// Mitsubishi GX Works2 project: 알람 터치스크린   PLC: Q02/Q02H

PROGRAM MAIN
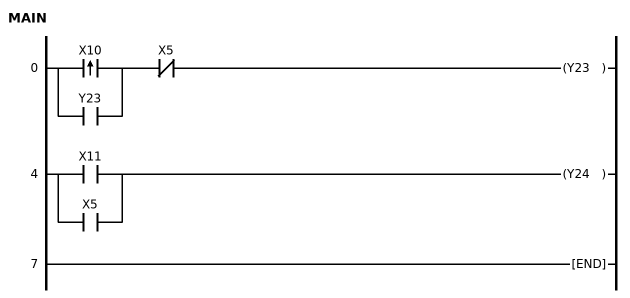
0     LDP     X10
      OR      Y23
      ANI     X5
      OUT     Y23
4     LD      X11
      OR      X5
      OUT     Y24
7     END
END_PROGRAM

PROGRAM HMI
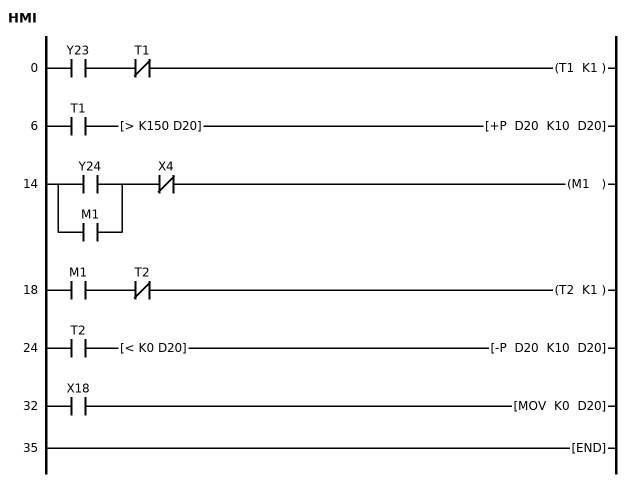
0     LD      Y23
      ANI     T1
      OUT     T1 K1
6     LD      T1
      AND>    K150 D20
      +P      D20 K10 D20
14    LD      Y24
      OR      M1
      ANI     X4
      OUT     M1
18    LD      M1
      ANI     T2
      OUT     T2 K1
24    LD      T2
      AND<    K0 D20
      -P      D20 K10 D20
32    LD      X18
      MOV     K0 D20
35    END
END_PROGRAM

PROGRAM ALARM
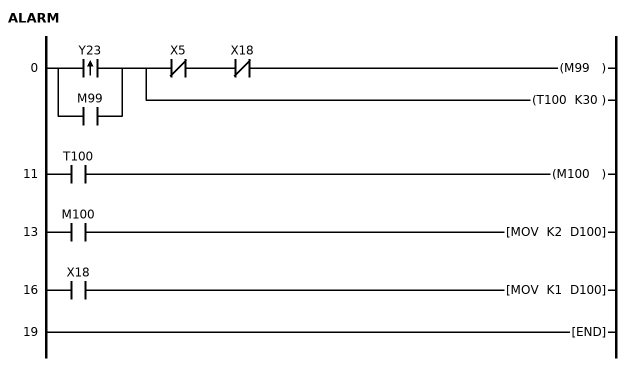
0     LDP     Y23
      OR      M99
      MPS
      ANI     X5
      ANI     X18
      OUT     M99
      MPP
      OUT     T100 K30
11    LD      T100
      OUT     M100
13    LD      M100
      MOV     K2 D100
16    LD      X18
      MOV     K1 D100
19    END
END_PROGRAM
